PROGRAM registradorLog20
VAR
	i: INT;
	j: INT;
	k: INT;
END_VAR


IF gvl.logRegister20 <> '' THEN
	FOR i:=100 TO 1 BY -1 DO
		IF gvl_p.arrLogEstufa20[i] <> '' THEN
			gvl_p.arrLogEstufa20[i+1]:= gvl_p.arrLogEstufa20[i];
			gvl_p.arrLogEstufa20[i]:= '';
		END_IF
	END_FOR
	gvl_p.arrLogEstufa20[1]:= concat(gvl_p.arrLogEstufa20[1],gvl.sSystemDateTime);
	gvl_p.arrLogEstufa20[1]:= concat(gvl_p.arrLogEstufa20[1],'    ');
	gvl_p.arrLogEstufa20[1]:= concat(gvl_p.arrLogEstufa20[1],gvl.logRegister20);
	gvl.sCmdInsertLog:= 'INSERT INTO [dbo].[LogGeneral] ([HistoricalTime],[Description])VALUES($'$',$'$')';
	gvl.sCmdInsertLog:= insert(gvl.sCmdInsertLog,gvl.logRegister20,74);	
	gvl.sCmdInsertLog:= insert(gvl.sCmdInsertLog,gvl.sSystemDateTime,71);
	gvl.bInsertLog:=true;
	gvl.logRegister20:= '';
	
	
END_IF

END_PROGRAM

(* stored: Version 1.1.0.1, ProductVersion 3.1.4024.12
   POU registradorLog20: Id {16095dbd-897e-44aa-b461-580ed1992e52}, SpecialFunc None *)
